// TIA Portal V20 export
DATA_BLOCK "DB_SonplasMain"   // DB88
// stored: InstanceOfName FB_SonplasMain, InstanceOfType FB
"FB_SonplasMain"
   // VAR
   //    sSonplasLoader : "FB_SonplasLoader";
   //    iDMC_CodeShuttle1 { S7_SetPoint := 'True'} : String;
   //    iDMC_CodeShuttle2 : String;
   //    iDMC_Code : String;
   //    oDMC_CodeShuttle1 : String;
   //    oDMC_CodeShuttle2 : String;
   //    oDMC_Code : String;
   // END_VAR
BEGIN
   sSonplasLoader.iPartInDMC_CodeShuttle1[0] := 16#0;
END_DATA_BLOCK
